FUNCTION_BLOCK FB_DriveMotion
VAR_INPUT
	iStart: BOOL; //TRUE to start the motion
	iInterlock: BOOL; //TRUE if the interlock is made
	iPowerOn:BOOL; //TRUE if the power is enabled on the station
	iManualMode: BOOL; //limit speed to 250mm/s
	iAutoCycling: BOOL; //auto mode
	iTargetPosn: LREAL; //target posn
	iMovetype: INT; //1= Abs, 2 = rel
	
	

END_VAR
VAR_OUTPUT
	qComplete: BOOL; //TRUE if the motion is complete
	qActive: BOOL; //TRUE if the motion is in progress

	

END_VAR
VAR
END_VAR

VAR_IN_OUT
	iqDriveInterface: typeDriveInterface;
	
END_VAR

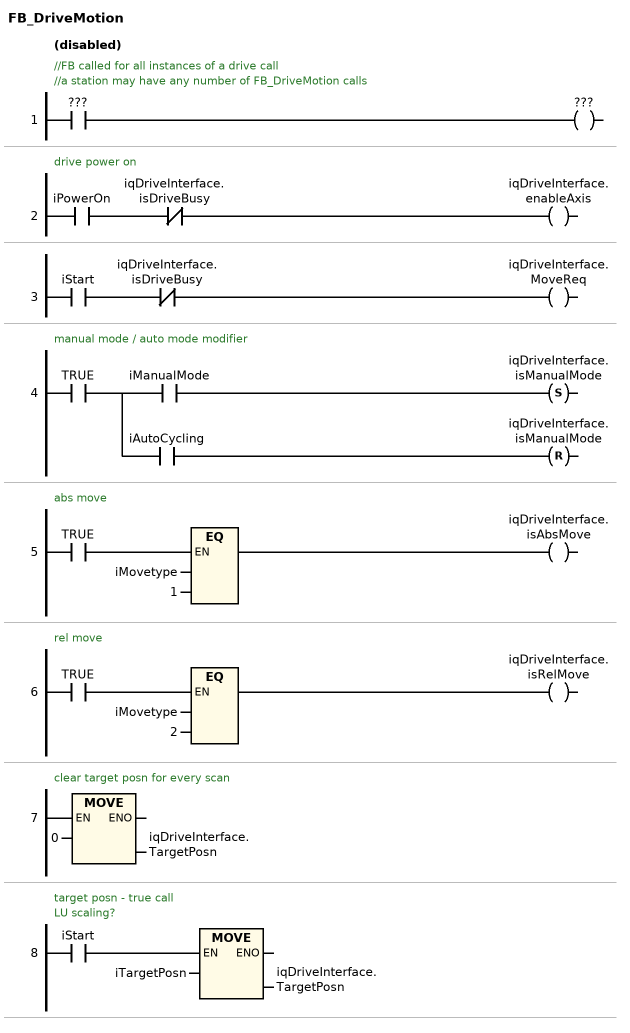
// NETWORK 1 (disabled)
// //FB called for all instances of a drive call
// //a station may have any number of FB_DriveMotion calls
// ??? := ???;

// NETWORK 2
// drive power on
iqDriveInterface.enableAxis := iPowerOn AND NOT iqDriveInterface.isDriveBusy;

// NETWORK 3
iqDriveInterface.MoveReq := iStart AND NOT iqDriveInterface.isDriveBusy;

// NETWORK 4
// manual mode / auto mode modifier
iqDriveInterface.isManualMode S= TRUE AND iManualMode;
iqDriveInterface.isManualMode R= TRUE AND iAutoCycling;

// NETWORK 5
// abs move
iqDriveInterface.isAbsMove := iMovetype = 1;

// NETWORK 6
// rel move
iqDriveInterface.isRelMove := iMovetype = 2;

// NETWORK 7
// clear target posn for every scan
iqDriveInterface.TargetPosn := 0;

// NETWORK 8
// target posn - true call
// LU scaling?
IF iStart THEN iqDriveInterface.TargetPosn := iTargetPosn; END_IF

END_FUNCTION_BLOCK

(* stored: Version 1.1.0.1, ProductVersion 3.1.4024.12
   POU FB_DriveMotion: Id {12882373-869e-456a-b6fe-dd0c072d47fc}, SpecialFunc None *)
